KUKA KRL program: dockon_2.src, dockon_2.dat

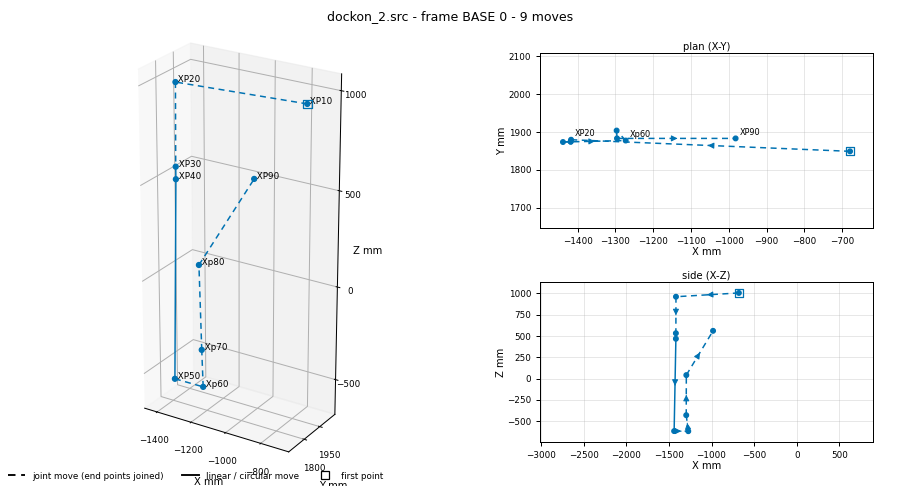
[picture p0: tool path of dockon_2.src in frame BASE 0, 9 of 9 moves have a stored position in this frame; points joined in program order, loops and branches not executed]
--- dockon_2.src ---
&ACCESS RV1
&REL 166
&COMMENT PICKUP  GUN 2
DEF DOCKON_2( )
;================================================
; MODEL    :
; IE GROUP :
; STATION  :
; ROBOT    :
; FUNCTION : DOCK ON GUN 2
;================================================
;FOLD INI
;FOLD BASISTECH INI
GLOBAL INTERRUPT DECL 3 WHEN $STOPMESS==TRUE DO IR_STOPM ( )
INTERRUPT ON 3
BAS (#INITMOV,0 )
;ENDFOLD (BASISTECH INI)
;FOLD USER INI
;Make your modifications here
;ENDFOLD (USER INI)
;ENDFOLD (INI)

;FOLD PTP p10  Vel= 100 % H Tool[10]:DOCKING PLATE Base[0];%{PE}%R 5.2.271,%MKUKATPBASIS,%CMOVE,%VPTP,%P 1:PTP, 2:p10, 3:, 5:100, 7:H
$BWDSTART = FALSE
PDAT_ACT=PH
FDAT_ACT=FP10
BAS(#PTP_PARAMS,100)
PTP XP10
;ENDFOLD

;Open flap 2
;FOLD DOCKING.FLAP_OPN 2 ;%{PE}%MKUKATPUSER
DOCKING (#FLAP_OPN ,2)
;ENDFOLD

;FOLD ; Check docking station 2 ready to dock on;%{PE}%R 2.4.14,%MKUKATPBASIS,%CCOMMENT,%VNORMAL,%P 2:Check docking station 2 ready to dock on
;ENDFOLD
DOCKING (#REQ_DOCK_ON ,2)

;FOLD PTP p20 CONT Vel= 100 % H Tool[10]:Docking plaat Base[0];%{PE}%R 5.2.271,%MKUKATPBASIS,%CMOVE,%VPTP,%P 1:PTP, 2:p20, 3:C_PTP, 5:100, 7:H
$BWDSTART = FALSE
PDAT_ACT=PH
FDAT_ACT=FP20
BAS(#PTP_PARAMS,100)
PTP XP20 C_PTP
;ENDFOLD

;FOLD ; Above dock position station 2;%{PE}%R 2.4.14,%MKUKATPBASIS,%CCOMMENT,%VNORMAL,%P 2:Above dock position station 2
;ENDFOLD
;FOLD PTP p30  Vel= 100 % H Tool[10]:Dock plate Base[0];%{PE}%R 5.4.35,%MKUKATPBASIS,%CMOVE,%VPTP,%P 1:PTP, 2:p30, 3:, 5:100, 7:H
$BWDSTART=FALSE
PDAT_ACT=PH
FDAT_ACT=FP30
BAS(#PTP_PARAMS,100)
PTP XP30
;ENDFOLD

;FOLD ; In Dock position Station 2;%{PE}%R 2.4.14,%MKUKATPBASIS,%CCOMMENT,%VNORMAL,%P 2:In Dock position Station 2
;ENDFOLD
;FOLD LIN p40  Vel= 0.2 m/s H Tool[10]:Dock plate Base[0];%{PE}%R 5.4.35,%MKUKATPBASIS,%CMOVE,%VLIN,%P 1:LIN, 2:p40, 3:, 5:0.2, 7:H
$BWDSTART=FALSE
LDAT_ACT=LH
FDAT_ACT=FP40
BAS(#CP_PARAMS,0.2)
LIN XP40
;ENDFOLD

;FOLD ; Lock Docking plate;%{PE}%R 2.4.14,%MKUKATPBASIS,%CCOMMENT,%VNORMAL,%P 2:Lock Docking plate
;ENDFOLD
DOCKING (#TOOL_LOCK ,2)

;FOLD ; Out Docking station 2;%{PE}%R 2.4.14,%MKUKATPBASIS,%CCOMMENT,%VNORMAL,%P 2:Out Docking station 2
;ENDFOLD
;FOLD LIN p50  Vel= 0.2 m/s H Tool[2]:Gun2 Base[0];%{PE}%R 5.4.35,%MKUKATPBASIS,%CMOVE,%VLIN,%P 1:LIN, 2:p50, 3:, 5:0.2, 7:H
$BWDSTART=FALSE
LDAT_ACT=LH
FDAT_ACT=FP50
BAS(#CP_PARAMS,0.2)
LIN XP50
;ENDFOLD

;FOLD ; Check docking plate close and station 2 ok;%{PE}%R 5.4.35,%MKUKATPBASIS,%CCOMMENT,%VNORMAL,%P 2:Check docking plate close and station 2 ok
;ENDFOLD
DOCKING (#CHK_TOOL_ON ,2)

;FOLD PTP p60  Vel= 30 % H Tool[2]:Gun2 Base[0];%{PE}%R 5.4.35,%MKUKATPBASIS,%CMOVE,%VPTP,%P 1:PTP, 2:p60, 3:, 5:30, 7:H
$BWDSTART=FALSE
PDAT_ACT=PH
FDAT_ACT=Fp60
BAS(#PTP_PARAMS,30)
PTP Xp60
;ENDFOLD
;FOLD PTP p70 CONT Vel= 100 % H Tool[2]:Gun2 Base[0];%{PE}%R 5.4.35,%MKUKATPBASIS,%CMOVE,%VPTP,%P 1:PTP, 2:p70, 3:C_PTP, 5:100, 7:H
$BWDSTART=FALSE
PDAT_ACT=PH
FDAT_ACT=Fp70
BAS(#PTP_PARAMS,100)
PTP Xp70 C_PTP
;ENDFOLD
;FOLD PTP p80 CONT Vel= 100 % H Tool[2]:Gun2 Base[0];%{PE}%R 5.4.35,%MKUKATPBASIS,%CMOVE,%VPTP,%P 1:PTP, 2:p80, 3:C_PTP, 5:100, 7:H
$BWDSTART=FALSE
PDAT_ACT=PH
FDAT_ACT=Fp80
BAS(#PTP_PARAMS,100)
PTP Xp80 C_PTP
;ENDFOLD
;FOLD PTP p90  Vel= 100 % H Tool[2]:Gun2 Base[0];%{PE}%R 5.4.35,%MKUKATPBASIS,%CMOVE,%VPTP,%P 1:PTP, 2:p90, 3:, 5:100, 7:H
$BWDSTART=FALSE
PDAT_ACT=PH
FDAT_ACT=FP90
BAS(#PTP_PARAMS,100)
PTP XP90
;ENDFOLD

END

--- dockon_2.dat ---
&ACCESS RV1
&REL 166
&COMMENT PICKUP  GUN 2
DEFDAT  DOCKON_2
;FOLD EXTERNAL DECLARATIONS;%{PE}%MKUKATPBASIS,%CEXT,%VCOMMON,%P
;FOLD GRIPPERTECH EXT
EXT  H50 (INT  :IN,INT  :IN,INT  :IN,GRP_TYP  :IN )
;ENDFOLD (GRIPPERTECH EXT)
;FOLD SPOTTECH EXT
EXT  USERSPOT (S_COMMAND  :IN,SPOT_TYPE  :IN )
;ENDFOLD (SPOTTECH EXT)
;FOLD BASISTECH EXT;%{PE}%MKUKATPBASIS,%CEXT,%VEXT,%P
EXT  BAS (BAS_COMMAND  :IN,REAL  :IN )
DECL INT SUCCESS
;ENDFOLD (BASISTECH EXT)
;FOLD USER EXT;%{E}%MKUKATPUSER,%CEXT,%VEXT,%P
;Make here your modifications
;ENDFOLD (USER EXT)
;ENDFOLD (EXTERNAL DECLERATIONS)
DECL GRP_TYP GCONT={G_APO #YES,TIME 0.0,CTRL #OFF,DLY 0,DST 0}
DECL GRP_TYP GGDAT={G_APO #NO,TIME 0.0,CTRL #OFF,DLY 0,DST 1}
;*      FDAT Declarations     *

;******************************
;*     E6POS Declarations     *
;******************************

DECL E6POS XP10={X -679.029297,Y 1849.03699,Z 1006.23798,A -155.054001,B -0.176167101,C -178.603394,S 2,T 43,E1 -735.491699,E2 0.0,E3 0.0,E4 0.0,E5 0.0,E6 0.0}
DECL E6POS XP20={X -1417.15295,Y 1879.72803,Z 961.852722,A -135.315201,B -0.308909208,C 179.562393,S 2,T 43,E1 -735.49353,E2 0.0,E3 0.0,E4 0.0,E5 0.0,E6 0.0}
DECL E6POS XP30={X -1418.18994,Y 1874.61597,Z 533.393921,A -134.240799,B -0.652091801,C 179.492203,S 2,T 43,E1 -735.497009,E2 0.0,E3 0.0,E4 0.0,E5 0.0,E6 0.0}
DECL E6POS XP40={X -1418.17505,Y 1874.60596,Z 468.598206,A -134.241104,B -0.651982188,C 179.492996,S 2,T 43,E1 -735.498779,E2 0.0,E3 0.0,E4 0.0,E5 0.0,E6 0.0}
DECL E6POS XP50={X -1438.63696,Y 1873.67505,Z -614.990112,A -84.244751,B -0.0316537693,C -0.824480712,S 2,T 43,E1 -735.49353,E2 0.0,E3 0.0,E4 0.0,E5 0.0,E6 0.0}
DECL E6POS XP60={X -1272.65906,Y 1877.58496,Z -616.231812,A -84.271347,B -0.0275246799,C -0.819864988,S 2,T 43,E1 -735.49353,E2 0.0,E3 0.0,E4 0.0,E5 0.0,E6 0.0}
DECL E6POS XP70={X -1296.66199,Y 1904.01196,Z -428.336792,A -85.3186111,B 0.148039997,C -0.629291892,S 2,T 43,E1 -735.491699,E2 0.0,E3 0.0,E4 0.0,E5 0.0,E6 0.0}
DECL E6POS XP80={X -1295.63403,Y 1883.23999,Z 42.0108414,A -85.3181534,B 0.148901105,C -0.630066872,S 2,T 43,E1 -735.491699,E2 0.0,E3 0.0,E4 0.0,E5 0.0,E6 0.0}
DECL E6POS XP90={X -981.813721,Y 1883.23096,Z 561.592896,A -85.3179092,B 0.148490995,C -0.62954849,S 2,T 43,E1 -735.49353,E2 0.0,E3 0.0,E4 0.0,E5 0.0,E6 0.0}

;******************************
;*     FDAT Declarations      *
;******************************

DECL FDAT FP10={TOOL_NO 10,BASE_NO 0,IPO_FRAME #BASE}
DECL FDAT FP20={TOOL_NO 10,BASE_NO 0,IPO_FRAME #BASE}
DECL FDAT FP30={TOOL_NO 10,BASE_NO 0,IPO_FRAME #BASE}
DECL FDAT FP40={TOOL_NO 10,BASE_NO 0,IPO_FRAME #BASE}
DECL FDAT FP50={TOOL_NO 2,BASE_NO 0,IPO_FRAME #BASE}
DECL FDAT FP60={TOOL_NO 2,BASE_NO 0,IPO_FRAME #BASE}
DECL FDAT FP70={TOOL_NO 2,BASE_NO 0,IPO_FRAME #BASE}
DECL FDAT FP80={TOOL_NO 2,BASE_NO 0,IPO_FRAME #BASE}
DECL FDAT FP90={TOOL_NO 2,BASE_NO 0,IPO_FRAME #BASE}

;******************************
;*  PDAT & LDAT Declarations  *
;******************************

DECL PDAT PH={VEL 100.0,ACC 100.0,APO_DIST 100.0}
DECL LDAT LH={VEL 2.0,ACC 100.0,APO_DIST 100.0,APO_FAC 50.0,ORI_TYP #VAR}

ENDDAT
